Omron Sysmac Studio project ShiftRotate (Sysmac Studio 1.65.0.64007, StandardProject)

# Controller new_Controller_0: NX1P2-1140DT1 version 1.69
Task PrimaryTask (priority 4, period or condition 2000): Program0



PROGRAM Program0
VAR
    trigger : BOOL;
    Ary1 : ARRAY[0..10] OF WORD;
    rst : BOOL;
    Inn : BOOL;
    ary2 : ARRAY[0..10] OF REAL;
    Data1 : WORD;
    RotatedData : WORD;
    Data2 : WORD;
    ShiftedData : WORD;
    AryShiftReg1 : AryShiftReg;
END_VAR
VAR
    _e1 : R_TRIG;
    _e2 : R_TRIG;
END_VAR

(* Section Section0: ladder, written here as Structured Text *)

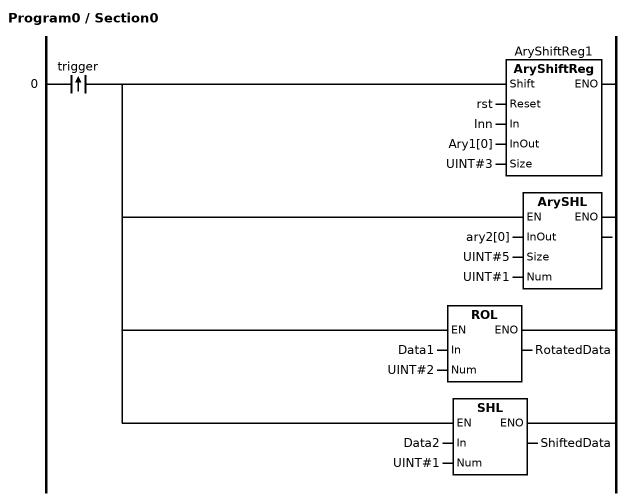
(* Rung 0 *)
_e1(CLK := trigger);
_e2(CLK := _e1.Q);
AryShiftReg1(Shift := _e2.Q, Reset := rst, In := Inn, InOut := Ary1[0], Size := UINT#3);
IF _e1.Q THEN
    ArySHL(InOut := ary2[0], Size := UINT#5, Num := UINT#1);
    RotatedData := ROL(In := Data1, Num := UINT#2);
    ShiftedData := SHL(In := Data2, Num := UINT#1);
END_IF;
END_PROGRAM